FUNCTION_BLOCK OnQueueChangedHandler EXTENDS OnQueueEventHandler

METHOD FB_init : BOOL
VAR_INPUT
	bInitRetains : BOOL; // if TRUE, the retain variables are initialized (warm start / cold start)
	bInCopyCode : BOOL;  // if TRUE, the instance afterwards gets moved into the copy code (online change)
	ExpectedOriginator : I_Queue;
END_VAR
SetExpectedOriginator(ExpectedOriginator);
END_METHOD

METHOD PUBLIC HandleEvent
VAR_INPUT
	Event : I_Event;
END_VAR
VAR
	queueChangedEvent : I_QueueChangedEvent;
END_VAR
IF __QUERYINTERFACE(Event, queueChangedEvent) THEN
	_eventReceived := TRUE;
	fromExpected := queueChangedEvent.TargetQueue = expectedOriginator;
END_IF
END_METHOD

METHOD PUBLIC SetExpectedOriginator
VAR_INPUT
	ExpectedOriginator : I_Queue;
END_VAR
this^.expectedOriginator := ExpectedOriginator;
END_METHOD

END_FUNCTION_BLOCK

(* stored: Version 1.1.0.1, ProductVersion 3.1.4024.12
   POU OnQueueChangedHandler: Id {32ce2bfe-57af-476b-9f9b-301331428837}, SpecialFunc None
   Folder Constructor: Id {5c606cc9-332d-440d-bc17-389e5de74fe5}
   Method FB_init: Id {adf32a6e-e697-4684-8e06-769bf531177e}
   Method HandleEvent: Id {d2734651-3c5c-45ee-b51c-4f93b9dd3f2f}
   Method SetExpectedOriginator: Id {eb79fbd6-3855-4955-bd72-2c7eb20fce75} *)
